// TIA Portal project "FactoryIO_Template_S7-1200_V16_V16" (V16)
// Vorlageprojekt für das Buch mit Zielsystem S7-1200

(* hardware
DEVICE "S7-1200-Station_1"  S7-1200 Station
   slot 0: "Baugruppenträger_0"  Rack  V1.0
   slot 1: "PLC_1"  CPU 1211C DC/DC/DC  6ES7 211-1AE40-0XB0  V4.1
*)

// ===== PLC "PLC_1"  CPU 1211C DC/DC/DC =====

VAR_GLOBAL   // PLC tag table "Standard-Variablentabelle"
   "conveyor 6" AT %A0.0 : Bool;
   "start" AT %E0.0 : Bool;
   "stop" AT %E0.1 : Bool;
   "Tag_4" AT %I10.0 : Bool;
   "Tag_5" AT %Q10.0 : Bool;
   "Tag_6" AT %I10.1 : Bool;
   "vision sensor 1" AT %I0.2 : Bool;
   "vision sensor 4" AT %I0.3 : Bool;
   "vision sensor 2" AT %I0.4 : Bool;
   "vision sensor 3" AT %I0.5 : Bool;
   "conveyor 1(2)" AT %Q0.1 : Bool;
   "conveyor 2(2)" AT %Q0.2 : Bool;
   "conveyor 3(2)" AT %Q0.3 : Bool;
   "conveyor 4(2)" AT %Q0.4 : Bool;
   "curved conveyor" AT %Q0.5 : Bool;
   "pivot arm 1" AT %Q0.6 : Bool;
   "pivot arm 1 belt" AT %Q0.7 : Bool;
   "pivot arm 2" AT %Q1.0 : Bool;
   "pivot arm 2 belt" AT %Q1.1 : Bool;
   "pivot arm 3" AT %Q1.2 : Bool;
   "pivot arm 3 belt" AT %Q1.3 : Bool;
   "Loop Marker" AT %M0.0 : Bool;
END_VAR

FUNCTION "MHJ-PLC-Lab-Function-S71200" : Void   // FC9000, SCL
{ S7_Optimized_Access := 'TRUE' }
VERSION : 0.1
   VAR_TEMP
      rdTimeReturn : Int;
      outputTime : DTL;
      SyncVal : Byte;
      forVal : Int;
      forVal_2 : Int;
      Value : Byte;
   END_VAR
   VAR CONSTANT
      CompVal : Byte := 16#34;
      Value_01 : Byte := 16#11;
      Value_01_DW : DWord := 16#A165_D992;
      Value_02_DW : DWord := 16#58BE_4401;
   END_VAR
BEGIN

   #Value:=PEEK(area := 16#82,
        dbNumber := 0,
        byteOffset := 511);
   #Value := #Value + 1;

   POKE(area := 16#82,
        dbNumber := 0,
        byteOffset := 511,
        value := #Value);

   POKE(area:=16#81,
        dbNumber:=0,
        byteOffset:=1016,
        value:=#Value_01_DW);
   POKE(area := 16#81,
        dbNumber := 0,
        byteOffset := 1020,
        value := #Value_02_DW);

   POKE(area := 16#81,
        dbNumber := 0,
        byteOffset := 511,
        value := B#16#00);

   FOR #forVal := 0 TO 120 DO
       FOR #forVal_2:=0 TO 10 DO
           #rdTimeReturn:=RD_SYS_T(#outputTime);
           #rdTimeReturn := WR_SYS_T(#outputTime);
           #rdTimeReturn := RD_SYS_T(#outputTime);
           #rdTimeReturn := WR_SYS_T(#outputTime);
       END_FOR;
       #SyncVal:= PEEK(area := 16#81,
                      dbNumber := 0,
                      byteOffset := 511);
       IF #SyncVal = #CompVal THEN
          GOTO M_1;
       END_IF;
   END_FOR;
   RETURN;

   M_1:
   POKE(area := 16#81,
        dbNumber := 0,
        byteOffset := 511,
        value := B#16#0);
END_FUNCTION

ORGANIZATION_BLOCK "Main"   // OB1, LAD, ProgramCycle
TITLE = "Main Program Sweep (Cycle)"
{ S7_Optimized_Access := 'TRUE' }
VERSION : 0.1
   VAR_INPUT
      Initial_Call : Bool;   // Initial call of this OB
      Remanence : Bool;   // =True, if remanent data are available
   END_VAR
BEGIN

REGION Network 1: Konnektierungsbaustein für PLC-Lab
   // Im Netzwerk 1 wird der Konnektierungsbaustein für PLC-Lab aufgerufen.
   // Dieser Aufruf darf nicht entfernt werden!
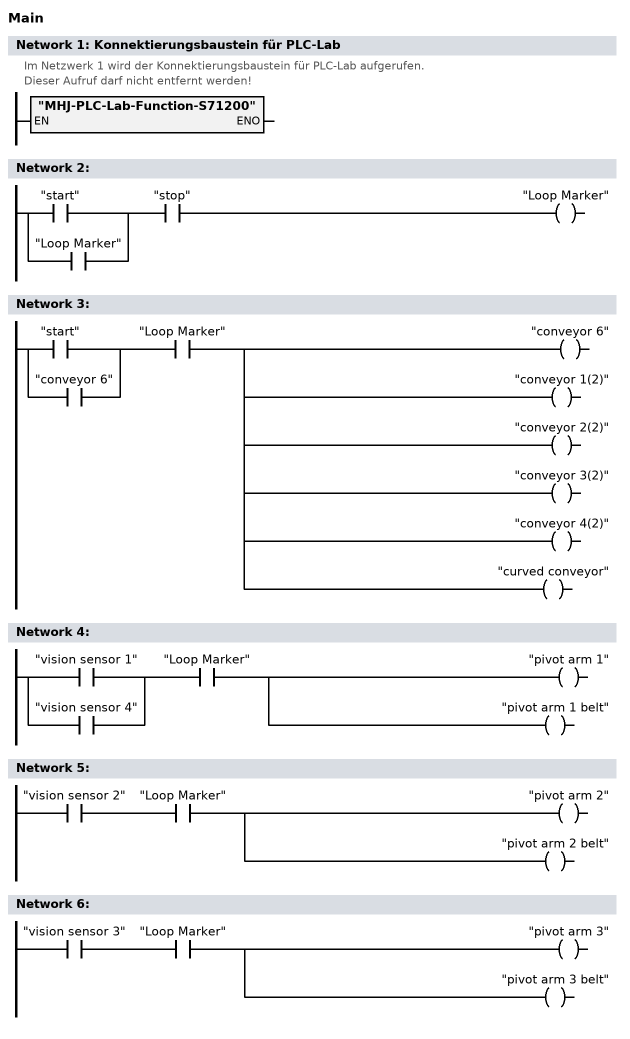
   RUNG wire#powerrail
      "MHJ-PLC-Lab-Function-S71200"()
   END_RUNG
   // the same network as SCL:
   "MHJ-PLC-Lab-Function-S71200"();
END_REGION

REGION Network 2
   RUNG wire#powerrail
      Contact( "start" )
      wire#w1
      Contact( "stop" )
      Coil( "Loop Marker" )
   END_RUNG
   RUNG wire#powerrail
      Contact( "Loop Marker" )
   END_RUNG wire#w1
   // the same network as SCL:
   "Loop Marker" := ("start" OR "Loop Marker") AND "stop";
END_REGION

REGION Network 3
   RUNG wire#powerrail
      Contact( "start" )
      wire#w1
      Contact( "Loop Marker" )
      wire#w2
      Coil( "conveyor 6" )
   END_RUNG
   RUNG wire#powerrail
      Contact( "conveyor 6" )
   END_RUNG wire#w1
   RUNG wire#w2
      Coil( "conveyor 1(2)" )
   END_RUNG
   RUNG wire#w2
      Coil( "conveyor 2(2)" )
   END_RUNG
   RUNG wire#w2
      Coil( "conveyor 3(2)" )
   END_RUNG
   RUNG wire#w2
      Coil( "conveyor 4(2)" )
   END_RUNG
   RUNG wire#w2
      Coil( "curved conveyor" )
   END_RUNG
   // the same network as SCL:
   "conveyor 6" := ("start" OR "conveyor 6") AND "Loop Marker";
   "conveyor 1(2)" := "conveyor 6";
   "conveyor 2(2)" := "conveyor 6";
   "conveyor 3(2)" := "conveyor 6";
   "conveyor 4(2)" := "conveyor 6";
   "curved conveyor" := "conveyor 6";
END_REGION

REGION Network 4
   RUNG wire#powerrail
      Contact( "vision sensor 1" )
      wire#w1
      Contact( "Loop Marker" )
      wire#w2
      Coil( "pivot arm 1" )
   END_RUNG
   RUNG wire#powerrail
      Contact( "vision sensor 4" )
   END_RUNG wire#w1
   RUNG wire#w2
      Coil( "pivot arm 1 belt" )
   END_RUNG
   // the same network as SCL:
   "pivot arm 1" := ("vision sensor 1" OR "vision sensor 4") AND "Loop Marker";
   "pivot arm 1 belt" := "pivot arm 1";
END_REGION

REGION Network 5
   RUNG wire#powerrail
      Contact( "vision sensor 2" )
      Contact( "Loop Marker" )
      wire#w1
      Coil( "pivot arm 2" )
   END_RUNG
   RUNG wire#w1
      Coil( "pivot arm 2 belt" )
   END_RUNG
   // the same network as SCL:
   "pivot arm 2" := "vision sensor 2" AND "Loop Marker";
   "pivot arm 2 belt" := "pivot arm 2";
END_REGION

REGION Network 6
   RUNG wire#powerrail
      Contact( "vision sensor 3" )
      Contact( "Loop Marker" )
      wire#w1
      Coil( "pivot arm 3" )
   END_RUNG
   RUNG wire#w1
      Coil( "pivot arm 3 belt" )
   END_RUNG
   // the same network as SCL:
   "pivot arm 3" := "vision sensor 3" AND "Loop Marker";
   "pivot arm 3 belt" := "pivot arm 3";
END_REGION
END_ORGANIZATION_BLOCK